{attribute 'linkalways'} 
{attribute 'no_explicit_call' := 'This FB is a CLASS and must be accessed using methods or properties'}
{attribute 'enable_dynamic_creation'}
FUNCTION_BLOCK FINAL OR_UINT EXTENDS Node
VAR
	in1 : _UINT(0);
	in2 : _UINT(0);
	out : _UINT(0);
END_VAR

METHOD PUBLIC Clone : I_Node
VAR
	pNode : POINTER TO OR_UINT;
END_VAR
pNode := __NEW(OR_UINT);
Clone := pNode^;
END_METHOD

METHOD FB_init : BOOL
VAR_INPUT
	bInitRetains : BOOL; // if TRUE, the retain variables are initialized (warm start / cold start)
	bInCopyCode : BOOL;  // if TRUE, the instance afterwards gets moved into the copy code (online change)
END_VAR
AddInput('in1',THIS^.in1);
AddInput('in2',THIS^.in2);
AddOutput('out', THIS^.out);
END_METHOD

METHOD PROTECTED OnExecute
VAR
END_VAR
out.Value := in1.Value OR in2.Value;
END_METHOD

END_FUNCTION_BLOCK

(* stored: Version 1.1.0.1, ProductVersion 3.1.4024.15
   POU OR_UINT: Id {96dee9bc-d598-459a-8b64-a4f9a57459bc}, SpecialFunc None
   Folder Constructor: Id {3cd9a0d6-52ac-4fad-84c3-cd0937f9058f}
   Method Clone: Id {3e65f880-c747-4225-8bf2-57e63d6cd94c}
   Method FB_init: Id {3fc2975f-b60e-43a6-a417-9224bdbfc1c7}
   Method OnExecute: Id {d4ed8596-ea83-432d-af59-7a4ccd00920b} *)
